PROGRAM sub_Access
VAR
	fbTuerGong		:	FB_Impulse;
	fbGaragentor	:	FB_Impulse;
END_VAR

//###################################################################################
//##-----------------------------------ACCESS--------------------------------------##
//###################################################################################

//--------------------TürGong----------------------------------
fbTuerGong.bInputs[0]	:= gvl_EA.bID24_01_1;

fbTuerGong(
	bR_Trig			:= TRUE,
	bInputSecLoop	:= gvl_mb.Output_Coils[245],
	bInputHA		:= gvl_mb.Output_Coils[14],
	tHigh			:= T#500MS,
	bOut			=> gvl_EA.bOD02_3
);
//-------------------------------------------------------------

//--------------------Garagentor----------------------------------
fbGaragentor.bInputs[0]	:= gvl_EA.bID05_1;

fbGaragentor(
	bR_Trig			:= TRUE,
	bInputHA		:= gvl_mb.Output_Coils[13],
	tHigh			:= T#500MS,
	bOut			=> gvl_EA.bWOD01_6
);
//-------------------------------------------------------------

END_PROGRAM

(* stored: Version 1.1.0.1, ProductVersion 3.1.4024.4
   POU sub_Access: Id {cf2eef73-b407-45a6-8d6e-b5c80300240a}, SpecialFunc None *)
